KUKA KRL program: spindle_main.src, spindle_main.dat

--- spindle_main.src ---
&ACCESS RVO
&REL 226
&PARAM EDITMASK = *
&PARAM TEMPLATE = C:\KRC\Roboter\Template\vorgabe
&PARAM DISKPATH = KRC:\R1\TP\Milling
DEF Spindle_MAIN()
;FOLD INI
  ;FOLD BASISTECH INI
    GLOBAL INTERRUPT DECL 3 WHEN $STOPMESS==TRUE DO IR_STOPM ( )
    INTERRUPT ON 3
    BAS (#INITMOV,0 )
  ;ENDFOLD (BASISTECH INI)
  ;FOLD USER INI
    ;Make your modifications here

  ;ENDFOLD (USER INI)
;ENDFOLD (INI)

PTP $AXIS_ACT

;FOLD PTP home Vel=100 % PDAT8;%{PE}%R 8.2.19,%MKUKATPBASIS,%CMOVE,%VPTP,%P 1:PTP, 2:home, 3:, 5:100, 7:PDAT8
$BWDSTART=FALSE
PDAT_ACT=PPDAT8
FDAT_ACT=Fhome
BAS(#PTP_PARAMS,100)
$H_POS=XHOME
PTP Xhome
;ENDFOLD
;FOLD MillingTech_Spindle_Function.SPINDLE_ENABLE SpindleOverride: blocked;%{PE}%MKUKATPUSER
Spindle_Enable(#blocked)
;ENDFOLD
;FOLD MillingTech_Air.SWITCH_MAINAIR_ON ;%{PE}%MKUKATPUSER
Air(#MainAirOn)
;ENDFOLD
;FOLD MillingTech_Chiller.SWITCH_ON ;%{PE}%MKUKATPUSER
Chiller(#ChillerOn)
;ENDFOLD


;FOLD MillingTech_Spindle_Function.ON Speed= 1000 rpm, Trigger: none, Offset: 0mm, Delay: 0 ms, Direction: clockwise;%{PE}%MKUKATPUSER
Spindle_Start(1000,#Standing,0,0,#CLOCKWISE)
;ENDFOLD



loop
;FOLD PTP home Vel=100 % PDAT4;%{PE}%R 8.2.19,%MKUKATPBASIS,%CMOVE,%VPTP,%P 1:PTP, 2:home, 3:, 5:100, 7:PDAT4
$BWDSTART=FALSE
PDAT_ACT=PPDAT4
FDAT_ACT=Fhome
BAS(#PTP_PARAMS,100)
$H_POS=XHOME
PTP Xhome
;ENDFOLD
;FOLD PTP p1 Vel=30 % PDAT5 Tool[1] Base[0];%{PE}%R 8.2.19,%MKUKATPBASIS,%CMOVE,%VPTP,%P 1:PTP, 2:p1, 3:, 5:30, 7:PDAT5
$BWDSTART=FALSE
PDAT_ACT=PPDAT5
FDAT_ACT=Fp1
BAS(#PTP_PARAMS,30)
PTP Xp1
;ENDFOLD


;FOLD PTP home Vel=30 % PDAT6;%{PE}%R 8.2.19,%MKUKATPBASIS,%CMOVE,%VPTP,%P 1:PTP, 2:home, 3:, 5:30, 7:PDAT6
$BWDSTART=FALSE
PDAT_ACT=PPDAT6
FDAT_ACT=Fhome
BAS(#PTP_PARAMS,30)
$H_POS=XHOME
PTP Xhome
;ENDFOLD
endloop
halt
;FOLD MillingTech_Spindle_Function.OFF Trigger: none, Offset: 0mm, Delay: 0 ms;%{PE}%MKUKATPUSER
Spindle_Stop(#Standing,0,0)
;ENDFOLD
halt

;FOLD MillingTech_Spindle_Function.SPINDLE_DISABLE ;%{PE}%MKUKATPUSER
Spindle_Disable()
;ENDFOLD
End

--- spindle_main.dat ---
&ACCESS RVO
&REL 226
&PARAM EDITMASK = *
&PARAM TEMPLATE = C:\KRC\Roboter\Template\vorgabe
&PARAM DISKPATH = KRC:\R1\TP\Milling
DEFDAT  spindle_main
;FOLD EXTERNAL DECLARATIONS;%{PE}%MKUKATPBASIS,%CEXT,%VCOMMON,%P
;FOLD BASISTECH EXT;%{PE}%MKUKATPBASIS,%CEXT,%VEXT,%P
EXT  BAS (BAS_COMMAND  :IN,REAL  :IN )
DECL INT SUCCESS
;ENDFOLD (BASISTECH EXT)
;FOLD USER EXT;%{E}%MKUKATPUSER,%CEXT,%VEXT,%P
;Make your modifications here

;ENDFOLD (USER EXT)
;ENDFOLD (EXTERNAL DECLARATIONS)
DECL BASIS_SUGG_T LAST_BASIS={POINT1[] "P2                      ",POINT2[] "P2                      ",CP_PARAMS[] "CPDAT0                  ",PTP_PARAMS[] "PDAT8                   ",CONT[] "                        ",CP_VEL[] "2.0                     ",PTP_VEL[] "30                      ",SYNC_PARAMS[] "SYNCDAT                 ",SPL_NAME[] "S0                      "}
DECL E6POS X$NULLFRAME={X 2053.66699,Y -241.348007,Z 1858.38904,A -170.6297,B 69.7047577,C -150.614594,S 2,T 34,E1 0.0,E2 0.0,E3 0.0,E4 0.0,E5 0.0,E6 0.0}
DECL FDAT F$nullframe={TOOL_NO 1,BASE_NO 0,IPO_FRAME #BASE,POINT2[] " ",TQ_STATE FALSE}
DECL PDAT PPDAT1={VEL 100.0,ACC 100.0,APO_DIST 100.0}
DECL PDAT PPDAT2={VEL 100.0,ACC 100.0,APO_DIST 100.0}
DECL PDAT PPDAT3={VEL 100.0,ACC 100.0,APO_DIST 100.0}
DECL PDAT PPDAT4={VEL 100.0,ACC 100.0,APO_DIST 100.0}
DECL E6POS XP1={X 1273.56104,Y -419.263306,Z 1808.89905,A -110.999397,B 86.321907,C -92.7864532,S 22,T 26,E1 0.0,E2 0.0,E3 0.0,E4 0.0,E5 0.0,E6 0.0}
DECL FDAT Fp1={TOOL_NO 1,BASE_NO 0,IPO_FRAME #BASE,POINT2[] " ",TQ_STATE FALSE}
DECL PDAT PPDAT5={VEL 100.0,ACC 100.0,APO_DIST 100.0}
DECL PDAT PPDAT6={VEL 100.0,ACC 100.0,APO_DIST 100.0}
DECL E6POS XP2={X 1431.31201,Y -531.325928,Z 1480.604,A -111.2985,B 86.3291092,C -93.075943,S 22,T 50,E1 0.0,E2 0.0,E3 0.0,E4 0.0,E5 0.0,E6 0.0}
DECL FDAT FP2={TOOL_NO 1,BASE_NO 0,IPO_FRAME #BASE,POINT2[] " ",TQ_STATE FALSE}
DECL PDAT PPDAT7={VEL 100.0,ACC 100.0,APO_DIST 100.0}
DECL PDAT PPDAT8={VEL 100.0,ACC 100.0,APO_DIST 100.0}
ENDDAT
